RoboDK station: Station.dk.rdk

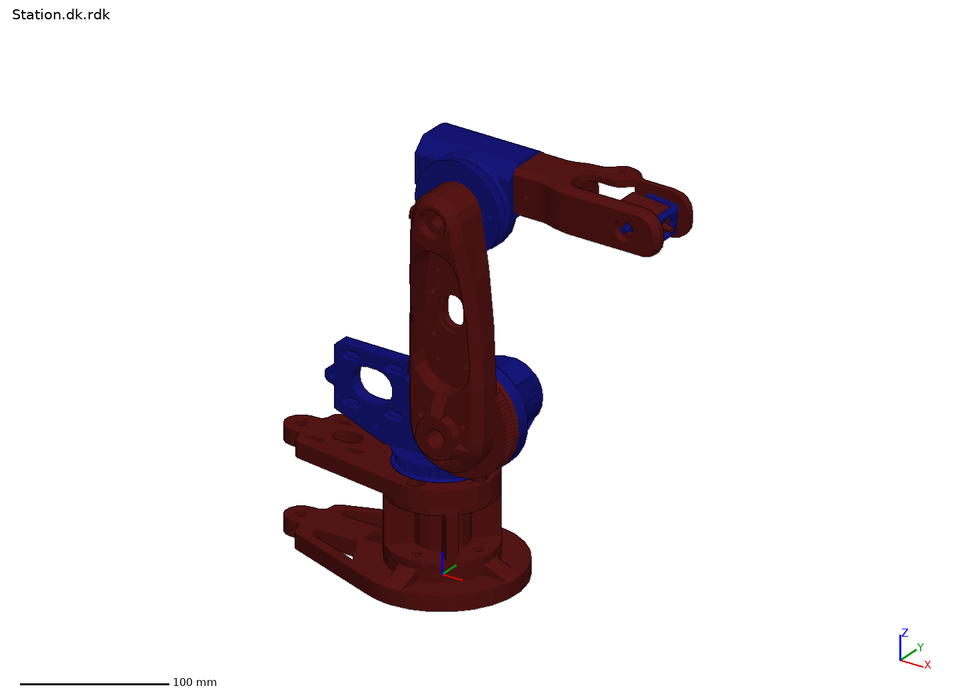
[picture v0: the station drawn from its stored meshes, robots at their saved joint values, targets as dots, program paths as lines]
Station Station.dk (saved by RoboDK 5.9.2). Poses are relative to the parent item; angles as X-Y-Z fixed-axis rotations.
  - frame My Mechanism Base at (145, 1015, 9) mm
    - robot My Mechanism: 6 axes
        modified DH rows (alpha deg, a mm, theta deg, d mm): 0, 0, 0, 135.3; -90, 37.5, -90, 0; 0, 160, 0, 0; -90, 15, 0, 137.3; 90, 0, 0, 0; -90, 0, 180, 0
        joint limits [-200, -80, -120, -200, -200, -200] to [200, 85, 65, 200, 200, 200]; home [0, 0, 0, 0, 0, 0]; saved at [0, 0, 0, 0, 0, 0]
